// TIA Portal V18 export
VAR_GLOBAL   // PLC tag table "Default tag table"
   Tag_2 AT %MD50 : Real;
   Tag_3 AT %M40.0 : Bool;
END_VAR
